# EPICS substitutions: bpmfeApp/Db/AKI2C_PCF85063TP.substitutions
file AKI2C_PCF85063TP_dev.template
{
   pattern { P    ,R    ,PORT    ,ADDR     ,TIMEOUT     }
           { $(P) ,$(R) ,$(PORT) ,$(ADDR)  ,$(TIMEOUT)  }
}
